(* PLC project TankLevelControl_LD, PLCAutoPilot Tank Level Control 1.0 *)
(* stored: creationDateTime 2025-12-25T12:00:00, modificationDateTime 2025-12-25T12:00:00 *)

(* Dual Tank Level Control Program - LADDER DIAGRAM VERSION RUNGS: 0 - System Start (Latch) 1 - System Stop 2 - Emergency Stop 3 - Pump 1 Command 4 - Pump 1 Output 5 - Pump 2 Command 6 - Pump 2 Output 7 - Running Light 8 - Tank 1 Low Alarm 9 - RO Tank Low Alarm 10 - Fault Detection OL1 11 - Fault Detection OL2 12 - Fault Light 13 - Fault Reset *)
PROGRAM Tank_Control_LD
  VAR
    System_Running : BOOL := FALSE;  (* System running flag *)
    Pump1_Cmd : BOOL := FALSE;
    Pump2_Cmd : BOOL := FALSE;
    Fault_Flag : BOOL := FALSE;
    Pump1_Timer : TON;
    Pump2_Timer : TON;
  END_VAR
  VAR_INPUT
    LS_Tank1 : BOOL;  (* Tank 1 Level Switch (0=Low, 1=High) *)
    LS_RO_Tank : BOOL;  (* RO Tank Level Switch (0=Low, 1=High) *)
    PB_Start : BOOL;  (* Start Push Button (NO) *)
    PB_Stop : BOOL;  (* Stop Push Button (NC) *)
    PB_EStop : BOOL;  (* Emergency Stop (NC) *)
    OL_Pump1 : BOOL;  (* Pump 1 Overload (NC) *)
    OL_Pump2 : BOOL;  (* Pump 2 Overload (NC) *)
  END_VAR
  VAR_OUTPUT
    Pump1_Out : BOOL;
    Pump2_Out : BOOL;
    Running_Light : BOOL;
    Tank1_Low_Alarm : BOOL;
    RO_Low_Alarm : BOOL;
    Fault_Light : BOOL;
  END_VAR

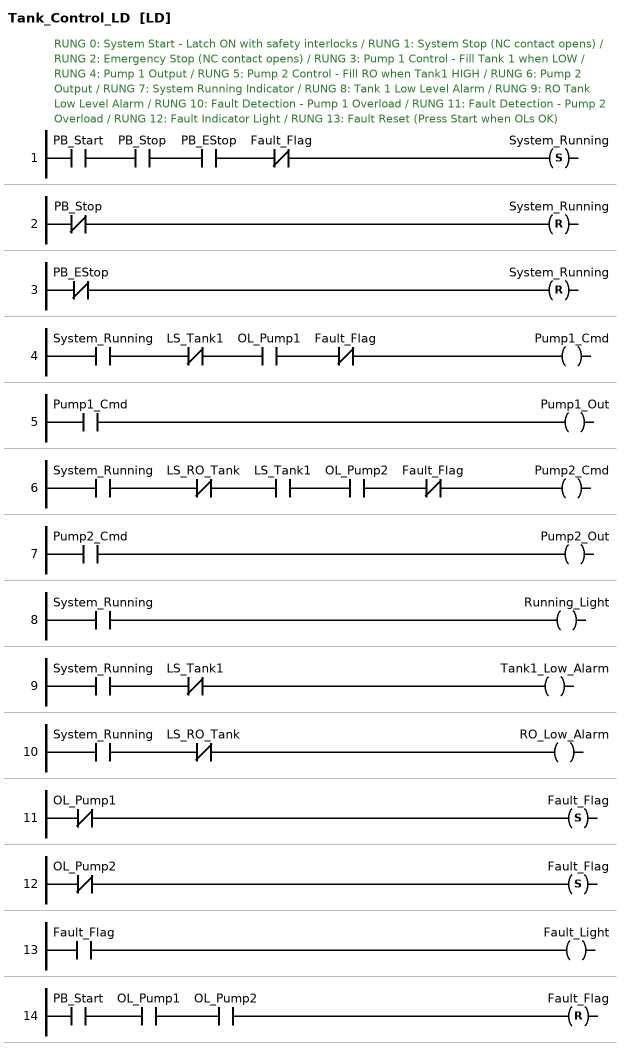
(* LD diagram, written out as Structured Text *)
(* RUNG 0: System Start - Latch ON with safety interlocks *)
IF PB_Start AND PB_Stop AND PB_EStop AND NOT Fault_Flag THEN System_Running := TRUE; END_IF;
(* RUNG 1: System Stop (NC contact opens) *)
IF NOT PB_Stop THEN System_Running := FALSE; END_IF;
(* RUNG 2: Emergency Stop (NC contact opens) *)
IF NOT PB_EStop THEN System_Running := FALSE; END_IF;
(* RUNG 3: Pump 1 Control - Fill Tank 1 when LOW *)
Pump1_Cmd := System_Running AND NOT LS_Tank1 AND OL_Pump1 AND NOT Fault_Flag;
(* RUNG 4: Pump 1 Output *)
Pump1_Out := Pump1_Cmd;
(* RUNG 5: Pump 2 Control - Fill RO when Tank1 HIGH *)
Pump2_Cmd := System_Running AND NOT LS_RO_Tank AND LS_Tank1 AND OL_Pump2 AND NOT Fault_Flag;
(* RUNG 6: Pump 2 Output *)
Pump2_Out := Pump2_Cmd;
(* RUNG 7: System Running Indicator *)
Running_Light := System_Running;
(* RUNG 8: Tank 1 Low Level Alarm *)
Tank1_Low_Alarm := System_Running AND NOT LS_Tank1;
(* RUNG 9: RO Tank Low Level Alarm *)
RO_Low_Alarm := System_Running AND NOT LS_RO_Tank;
(* RUNG 10: Fault Detection - Pump 1 Overload *)
IF NOT OL_Pump1 THEN Fault_Flag := TRUE; END_IF;
(* RUNG 11: Fault Detection - Pump 2 Overload *)
IF NOT OL_Pump2 THEN Fault_Flag := TRUE; END_IF;
(* RUNG 12: Fault Indicator Light *)
Fault_Light := Fault_Flag;
(* RUNG 13: Fault Reset (Press Start when OLs OK) *)
IF PB_Start AND OL_Pump1 AND OL_Pump2 THEN Fault_Flag := FALSE; END_IF;
END_PROGRAM

CONFIGURATION TankControl_Config
  RESOURCE TankControl_Resource ON PLC
    TASK MAST(INTERVAL := T#10ms, PRIORITY := 1);
    PROGRAM Tank_Control_LD_Instance WITH MAST : Tank_Control_LD;
  END_RESOURCE
END_CONFIGURATION
